FUNCTION_BLOCK ABSTRACT FB_Test2 EXTENDS FB_Test1_Base IMPLEMENTS I_Base
VAR_INPUT
  i : INT;
END_VAR
VAR_OUTPUT
END_VAR
VAR
END_VAR

{warning 'Methodenimplementierung hinzufügen'}
/// This is a TestMethod
METHOD M_Test1 : INT
END_METHOD

METHOD M_Test2 : BOOL
VAR_INPUT
END_VAR
END_METHOD

{warning 'Eigenschaftenimplementierung hinzufügen'}
(* A Test Property with get and set*)
PROPERTY P_TestFor : BOOL
GET
END_GET
SET
END_SET
END_PROPERTY

END_FUNCTION_BLOCK

(* stored: Version 1.1.0.1
   POU FB_Test2: Id {75ba6874-2021-49a5-8686-502a27f69b48}, SpecialFunc None
   Method M_Test1: Id {c0d66810-7824-4783-8c39-d5b5c2e2e780}
   Method M_Test2: Id {fabd59d4-8007-488b-8c84-a98a80d764d0}
   Property P_TestFor: Id {55148c74-7c9f-4698-ae73-8b45e389e590}
   Get Get: Id {736795d1-82c0-40d6-97d8-2d7d528a811e}
   Set Set: Id {1c063c5d-338a-4a83-a19b-cede26bba8de} *)
